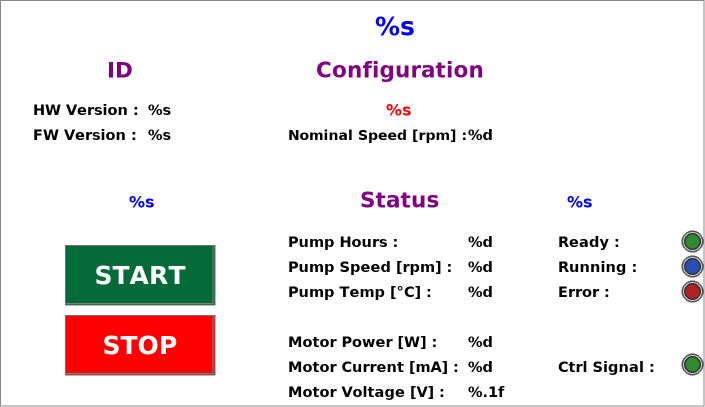
VISUALIZATION GUI_TEMPLATE_MVP030  // 705x407
VAR_IN_OUT
	m_Instance:	FB_CRYO_PUMP_MVP030;
	m_bEnable:	BOOL;	// Flag to start/stop the pump
END_VAR
    Rectangle (45,55 150x30), "ID"
    Rectangle (310,55 180x30), "Configuration"
    Rectangle (325,185 150x30), "Status"
    Lamp1 (680,229 25x25), tooltip "OK for Process, i.e. speed ≥ nominal speed", variable: m_Instance.stat.bReady, style: Lamp-Lamp1-Green
    Lamp1 (680,254 25x25), tooltip "pump speed > 0 rpm", variable: m_Instance.stat.bMoving, style: Lamp-Lamp1-Blue
    Lamp1 (680,279 25x25), tooltip "presence of a warning", variable: m_Instance.stat.bFailure, style: Lamp-Lamp1-Red
    Rectangle (555,227 110x30), "Ready :"
    Rectangle (555,252 110x30), "Running :"
    Rectangle (555,277 110x30), "Error :"
    Rectangle (285,120 180x30), "Nominal Speed [rpm] :"
    Rectangle (285,227 180x30), "Pump Hours :"
    Rectangle (465,120 70x30), "%d", text variable: m_Instance.stat.nNominalSpeed
    Rectangle (465,227 70x30), "%d", text variable: m_Instance.stat.nPumpHours
    Rectangle (285,252 180x30), "Pump Speed [rpm] :"
    Rectangle (465,252 70x30), "%d", text variable: m_Instance.stat.nPumpSpeed
    Rectangle (285,277 180x30), "Pump Temp [°C] :"
    Rectangle (465,277 70x30), "%d", text variable: m_Instance.stat.nPumpTemp
    Rectangle (285,352 180x30), "Motor Current [mA] :"
    Rectangle (465,352 70x30), "%d", text variable: m_Instance.stat.nMotorCurr
    Rectangle (285,377 180x30), "Motor Voltage [V] :"
    Rectangle (465,377 70x30), "%.1f", text variable: m_Instance.stat.lrMotorVolt
    Rectangle (280,11 230x30), "%s", text variable: m_Instance.in_sName
    Rectangle (289,95 220x30), "%s", tooltip "Control Mode", text variable: m_Instance.stat.sCtrlMode
    Rectangle (145,95 130x30), "%s", tooltip "HW Version", text variable: m_Instance.stat.sHwVersion
    Rectangle (145,120 130x30), "%s", tooltip "FW Version", text variable: m_Instance.stat.sFwVersion
    Button (65,245 150x60), "START"
        OnMouseClick: execute { m_bEnable := TRUE; }
    Button (65,315 150x60), "STOP"
        OnMouseClick: execute { m_bEnable := FALSE; }
    Lamp1 (680,352 25x25), tooltip "If ON, control output signal is active.", variable: m_Instance.q_bStart, style: Lamp-Lamp1-Green
    Rectangle (555,352 110x30), "Ctrl Signal :"
    Rectangle (457,187 246x30), "%s", tooltip "Pump State", text variable: m_Instance.stat.sPumpState
    Rectangle (92,187 100x30), "%s", tooltip "Error Status", text variable: m_Instance.stat.sFailureCode
    Rectangle (285,327 180x30), "Motor Power [W] :"
    Rectangle (465,327 70x30), "%d", text variable: m_Instance.stat.nElecPower
    Rectangle (30,95 110x30), "HW Version :"
    Rectangle (30,120 110x30), "FW Version :"
END_VISUALIZATION

(* stored: Version 1.1.0.1, ProductVersion 3.1.4024.12
   Visu GUI_TEMPLATE_MVP030: Id {a176ad9a-1f1d-4d06-ab8c-37903ad69e98} *)
